FUNCTION_BLOCK FB_A_HKSystem
VAR_INPUT
	I_bVerbunden	:BOOL;		// Angabe ob HK-System angeschlossen ist
	I_iModus		:INT;		// Zustand des Systems (z.B. 0 = AUS | 1 = MAN | 2 = AUTO)
	I_bVerriegeln	:BOOL;		// Verriegelte Elemente sind nicht ansteuerbar
	I_iTemp			:INT;		// Angabe der aktuellen Temperatur
	I_bReset		:BOOL;		// Zustand des Baustein wird zurückgesetzt 
END_VAR

VAR_OUTPUT
	O_bKuehlen		:BOOL;		// HK-System heizt das Medium auf
	O_bHeizen		:BOOL;		// HK-System kühlt das Medium ab
	O_bError		:BOOL;		// Befindet sich das Element in einem Error
	O_iStoerungID	:INT;		// Anzeigen von Störung über eine INT-Variable
	
END_VAR
	
VAR
	V_TempMax		:INT;		// Variable für internes handling der Eigenschaft 
	V_TempMin		:INT;		// Variable für internes handling der Eigenschaft 
	V_Zustand		:INT;		// Variable für internes handling der Eigenschaft 
END_VAR

METHOD M_A_HEIZEN : BOOL
VAR_INPUT
END_VAR
END_METHOD

METHOD M_A_KUEHLEN : BOOL
VAR_INPUT
END_VAR
END_METHOD

METHOD M_M_HEIZEN : BOOL
VAR_INPUT
END_VAR
END_METHOD

METHOD M_M_KUEHLEN : BOOL
VAR_INPUT
END_VAR
END_METHOD

PROPERTY PUBLIC P_MaxTemp : INT
SET
END_SET
END_PROPERTY

PROPERTY PUBLIC P_MinTemp : INT
SET
END_SET
END_PROPERTY

PROPERTY PUBLIC P_Zustand : INT
GET
END_GET
END_PROPERTY

END_FUNCTION_BLOCK

(* stored: Version 1.1.0.1, ProductVersion 3.1.4024.12
   POU FB_A_HKSystem: Id {9fa8220f-7562-4362-b973-7f9818c39521}, SpecialFunc None
   Method M_A_HEIZEN: Id {805f7cbf-a553-4d3b-9434-906e69543a3f}
   Method M_A_KUEHLEN: Id {553ba116-732f-49c2-828c-c4f64984a7f1}
   Method M_M_HEIZEN: Id {9431c962-da2e-4e6c-85e5-1e6aa4bd1568}
   Method M_M_KUEHLEN: Id {edd300d5-3c05-4015-826d-b28d4c741cb4}
   Property P_MaxTemp: Id {087eb6ba-a3ae-4a3e-a81a-2c88e8429d48}
   Set Set: Id {57e4acaf-0195-44c0-aea7-370b573f2cfb}
   Property P_MinTemp: Id {bfb56a72-03b9-4009-b5d0-39b88f56029f}
   Set Set: Id {810a7e51-bfb0-4f98-8bdb-2701d93499dd}
   Property P_Zustand: Id {41e75813-f874-43a5-bfc6-f44385e63ae2}
   Get Get: Id {49cb2351-eb2a-4219-9220-c46d74796b7d} *)
